(********************************************************************************************)
(*							Beckhoff Automation Poland										*)
(*								FB_XCopyCE  v1.0											*)
(*									07.07.2010												*)
(*	Bloczek kopiujący plik z miejsca zrodlowego do docelowego,  							*)
(*	jesli w miejscu docelowym jest juz plik o tej nazwie, zostanie on zastąpiony			*)
(*	BF wykorzystuje  NT_StartProcess znajudjący się w bibliotece TcUtilities.lib			*)
(*	Sprawdzony pod systemem Windows CE5 i CE6, wymaga pliku 	\Hard Disk\System\XCOPYCE	*)
(*__________________________________________________________________________________________*)
FUNCTION_BLOCK FB_XCopyCE
VAR_INPUT
	bCopy : 			BOOL;	(* zbocze narastajace rozpoczyna kopiowanie *)
	NetID: 				STRING;
	sFileName : 		STRING;	(* nazwa pliku np: 'a.txt' *)
	sSrcPath : 			STRING;	(* sciezka zrodlowa np: '\Hard Disk\' *)
	sDestPath :		 	STRING;	(* sciezka docelowa np: '\Hard Disk\ftp\' *)

END_VAR
VAR_OUTPUT
	bBusy : 			BOOL;
	bError :	 		BOOL;
	bErrID :			UDINT;
END_VAR
VAR
	NtStartProcess : 	NT_StartProcess;
	rtCopy: 			R_TRIG;
	step: 				INT;
	sCmd: 				STRING;
END_VAR

rtCopy(CLK:= bCopy, Q=> );

IF rtCopy.Q THEN 	step := step +10; END_IF

CASE step OF
0:	(* czeka na polecenie kopiowania *)
	bBusy:= FALSE;
	NtStartProcess.START := FALSE;
10:
	bBusy := TRUE;
	bError := FALSE;
	bErrID :=0;
	sCmd:='';				(* tworzenie polecenia *)
	sCmd := CONCAT(CONCAT(CONCAT('"', sSrcPath), sFileName), '" "');
	sCmd := CONCAT(CONCAT(sCmd, sDestPath), '" /Y');
	NtStartProcess.START := TRUE;
	step := step +10;

20:
	IF NOT NtStartProcess.BUSY AND NOT NtStartProcess.ERR THEN
		step := Step -20;
	ELSIF  NtStartProcess.ERR THEN
		Step := step -20;
		bError := TRUE;
		bErrID := NtStartProcess.ERRID;
	END_IF
END_CASE



NtStartProcess(
	NETID:= NetID,
	PATHSTR:=  '\Hard Disk\System\XCOPYCE',
	DIRNAME:=  '\Hard Disk\System',
	COMNDLINE:= sCmd ,
	START:= ,
	TMOUT:= ,
	BUSY=> ,
	ERR=> , 
	ERRID=> );

END_FUNCTION_BLOCK

(* stored: Version 1.1.0.1, ProductVersion 3.1.4020.3
   POU FB_XCopyCE: Id {6d862a1b-3920-4370-bfec-6b7601462589}, SpecialFunc None *)
